// TIA Portal V20 export
DATA_BLOCK "EncoderTel81"   // DB44
{ S7_Optimized_Access := 'FALSE' }
   VAR
      Tel81 { S7_SetPoint := 'True'} : PD_TEL81;
   END_VAR
BEGIN
END_DATA_BLOCK
